// TIA Portal V20 export
DATA_BLOCK "HMI_DB"   // DB15
{ S7_Optimized_Access := 'TRUE' }
// stored: MemoryReserve 100
   VAR
      ActiveScreenName : String;
      Tip_MT_Control : Bool;
      Tip_HMI_Control : Bool;
      Tip_Up : Bool;
      Tip_Down : Bool;
      TipMT_Arm_Selection : Int;
      TipMT_Button_Up : Bool;
      TipMT_Button_Down : Bool;
      TipMT_Set_Angle : Int;
      TipMT_Button_Open : Bool;
      TipMT_Button_Close : Bool;
      Safety_ACK : Bool;
      Reset_Drives : Bool;
      Reset_Safety : Bool;
      Reset_Reinicialisation : Bool;
      CNTUp : Bool;
      CNTDown : Bool;
      Heart_Bit : USInt;
   END_VAR
BEGIN
END_DATA_BLOCK
